PROGRAM prgMotionRow
VAR
		tStationNumberIndex: UINT;	
		tNumElementsPerScreen: UINT;
		tScreenElementsPerPage: UINT;
		tTrueStationIndex: UINT;
		tSizeOfMotionRow: UINT;
		tSizeOfMotionRowButtons: UINT;
		retval: UDINT;
		btnNext:R_TRIG;
		btnPrev:R_TRIG;
		
		btnNextRow:R_TRIG;
		btnPrevRow:R_TRIG;
		tSingleRowOffset: UINT;
		
	tSingleRowOffsettest: UINT;
	tSingleRowOffsettestbtns: UINT;
	tSizeOfButtonsLen: UINT;
	tSizeOfRowSingleLens: UINT;
	
	tSingleRowOffsetFactor:UINT;
	tSingleRowOffsetPointer: UINT;
END_VAR

//call logic for Motion screen using motion Rows

//select station on HMI
actPageControl();

//calculate screen range
actCalcScreenNumber();

//call manual screen rows
actCallMotionScreen();

//calculate screen range
actCalcMotionRowPosn();

//calculate page title
actCalcPageTitle();

ACTION actCalcMotionRowPosn:
//calaculate station index for pages
tTrueStationIndex := tStationNumberIndex + ((tScreenElementsPerPage * gHMIData.gActivePageNumber) -  tScreenElementsPerPage);


tSingleRowOffsetPointer := (tSingleRowOffsetFactor *  gHMIDataConst.gNumberElementsPerRow) - gHMIDataConst.gNumberElementsPerRow;
tSingleRowOffsetPointer := tSingleRowOffsetPointer + gHMIDataConst.gNumberElementsPerRow;

//test for singular row change
tTrueStationIndex := tTrueStationIndex + tSingleRowOffsetPointer;

//calculate offset for row x
gHMIData.gRowElementOffset[1]:= tTrueStationIndex + ((gHMIDataConst.gNumberElementsPerRow * 1) - gHMIDataConst.gNumberElementsPerRow);
gHMIData.gRowElementOffset[2]:= tTrueStationIndex + ((gHMIDataConst.gNumberElementsPerRow * 2) - gHMIDataConst.gNumberElementsPerRow);
gHMIData.gRowElementOffset[3]:= tTrueStationIndex + ((gHMIDataConst.gNumberElementsPerRow * 3) - gHMIDataConst.gNumberElementsPerRow);
gHMIData.gRowElementOffset[4]:= tTrueStationIndex + ((gHMIDataConst.gNumberElementsPerRow * 4) - gHMIDataConst.gNumberElementsPerRow);
gHMIData.gRowElementOffset[5]:= tTrueStationIndex + ((gHMIDataConst.gNumberElementsPerRow * 5) - gHMIDataConst.gNumberElementsPerRow);
gHMIData.gRowElementOffset[6]:= tTrueStationIndex + ((gHMIDataConst.gNumberElementsPerRow * 6) - gHMIDataConst.gNumberElementsPerRow);
gHMIData.gRowElementOffset[7]:= tTrueStationIndex + ((gHMIDataConst.gNumberElementsPerRow * 7) - gHMIDataConst.gNumberElementsPerRow);
gHMIData.gRowElementOffset[8]:= tTrueStationIndex + ((gHMIDataConst.gNumberElementsPerRow * 8) - gHMIDataConst.gNumberElementsPerRow);
gHMIData.gRowElementOffset[9]:= tTrueStationIndex + ((gHMIDataConst.gNumberElementsPerRow * 9) - gHMIDataConst.gNumberElementsPerRow);


//move to global to be picked up by each row
gHMIMotionRows.gMotionRows.gMotionRow1.IndexLocation := gHMIData.gRowElementOffset[1];
gHMIMotionRows.gMotionRows.gMotionRow2.IndexLocation := gHMIData.gRowElementOffset[2];
gHMIMotionRows.gMotionRows.gMotionRow3.IndexLocation := gHMIData.gRowElementOffset[3];
gHMIMotionRows.gMotionRows.gMotionRow4.IndexLocation := gHMIData.gRowElementOffset[4];
gHMIMotionRows.gMotionRows.gMotionRow5.IndexLocation := gHMIData.gRowElementOffset[5];
gHMIMotionRows.gMotionRows.gMotionRow6.IndexLocation := gHMIData.gRowElementOffset[6];
gHMIMotionRows.gMotionRows.gMotionRow7.IndexLocation := gHMIData.gRowElementOffset[7];
gHMIMotionRows.gMotionRows.gMotionRow8.IndexLocation := gHMIData.gRowElementOffset[8];
gHMIMotionRows.gMotionRows.gMotionRow9.IndexLocation := gHMIData.gRowElementOffset[9];
END_ACTION

ACTION actCalcPageTitle:
//get the page number index relating the group of motions displayed
gHMIData.gManualScreenTitle := tStationNumberIndex + gHMIData.gActivePageNumber;

//10001 = station 1, page 1
//10002 = station 1, page 2

//20001 = station 1, page 1
//etc

//assign text in textlist ManualPageTitle
END_ACTION

ACTION actCalcScreenNumber:
//create number for station
tStationNumberIndex := gHMIData.gActiveStationNumber * 10000;

//calculate number of elements per screen
tNumElementsPerScreen := gHMIDataConst.gNumberRowsPerPage * gHMIDataConst.gNumberElementsPerRow;

//calculate screen per page index
tScreenElementsPerPage := tNumElementsPerScreen  * 1;
END_ACTION

ACTION actCallMotionScreen:
//calculate byte offset - motions
tSizeOfMotionRow		:= gHMIData.gActivePageNumber * SIZEOF(gHMIMotionRows.gMotionRows);
tSizeOfMotionRow 		:= tSizeOfMotionRow - SIZEOF(gHMIMotionRows.gMotionRows);

//test for singular row changes
tSizeOfRowSingleLens := SIZEOF(typeMotionRow); //typ 153 bytes
tSizeOfMotionRow := tSizeOfMotionRow + (tSingleRowOffsetFactor * tSizeOfRowSingleLens) ;


//calculate byte offset - buttons
tSizeOfMotionRowButtons := gHMIData.gActivePageNumber * SIZEOF(gHMIMotionRows.gMotionRowButtons);
tSizeOfMotionRowButtons := tSizeOfMotionRowButtons - SIZEOF(gHMIMotionRows.gMotionRowButtons);

//test for singular row changes
tSizeOfButtonsLen := SIZEOF(typeMotionRowButtons); // typ 83 bytes
tSizeOfMotionRowButtons := tSizeOfMotionRowButtons + (tSingleRowOffsetFactor * tSizeOfButtonsLen);

//move data based on station and page number
//Move feedback indicator data
//Move Button BOOL state back adr(S1_Global.MotionRow)
IF gHMIData.gStationSelected[1] THEN
	retval := memcpy(	destAddr:=	ADR(gHMIMotionRows.gMotionRows),
						srcAddr:=	ADR(S1_Global.station.MotionRow) + tSizeOfMotionRow,
						n:=			SIZEOF(gHMIMotionRows.gMotionRows)
						);
						
	retval := memcpy(	destAddr:=	ADR(S1_Global.station.MotionRowBtn) + tSizeOfMotionRowButtons,
						srcAddr:=	ADR(gHMIMotionRows.gMotionRowButtons),
						n:=			SIZEOF(gHMIMotionRows.gMotionRowButtons)
						);
END_IF

IF gHMIData.gStationSelected[2] THEN
	retval := memcpy(	destAddr:=	ADR(gHMIMotionRows.gMotionRows),
						srcAddr:=	ADR(S2_Global.station.MotionRow) + tSizeOfMotionRow,
						n:=			SIZEOF(gHMIMotionRows.gMotionRows)
						);
						
	retval := memcpy(	destAddr:=	ADR(S2_Global.station.MotionRowBtn) + tSizeOfMotionRowButtons,
						srcAddr:=	ADR(gHMIMotionRows.gMotionRowButtons),
						n:=			SIZEOF(gHMIMotionRows.gMotionRowButtons)
						);
END_IF

IF gHMIData.gStationSelected[3] THEN
	retval := memcpy(	destAddr:=	ADR(gHMIMotionRows.gMotionRows),
						srcAddr:=	ADR(S3_Global.station.MotionRow) + tSizeOfMotionRow,
						n:=			SIZEOF(gHMIMotionRows.gMotionRows)
						);
						
	retval := memcpy(	destAddr:=	ADR(S3_Global.station.MotionRowBtn) + tSizeOfMotionRowButtons,
						srcAddr:=	ADR(gHMIMotionRows.gMotionRowButtons),
						n:=			SIZEOF(gHMIMotionRows.gMotionRowButtons)
						);
END_IF

IF gHMIData.gStationSelected[4] THEN
	retval := memcpy(	destAddr:=	ADR(gHMIMotionRows.gMotionRows),
						srcAddr:=	ADR(S4_Global.station.MotionRow) + tSizeOfMotionRow,
						n:=			SIZEOF(gHMIMotionRows.gMotionRows)
						);
						
	retval := memcpy(	destAddr:=	ADR(S4_Global.station.MotionRowBtn) + tSizeOfMotionRowButtons,
						srcAddr:=	ADR(gHMIMotionRows.gMotionRowButtons),
						n:=			SIZEOF(gHMIMotionRows.gMotionRowButtons)
						);
END_IF

IF gHMIData.gStationSelected[5] THEN
	retval := memcpy(	destAddr:=	ADR(gHMIMotionRows.gMotionRows),
						srcAddr:=	ADR(S5_Global.station.MotionRow) + tSizeOfMotionRow,
						n:=			SIZEOF(gHMIMotionRows.gMotionRows)
						);
						
	retval := memcpy(	destAddr:=	ADR(S5_Global.station.MotionRowBtn) + tSizeOfMotionRowButtons,
						srcAddr:=	ADR(gHMIMotionRows.gMotionRowButtons),
						n:=			SIZEOF(gHMIMotionRows.gMotionRowButtons)
						);
END_IF

IF gHMIData.gStationSelected[6] THEN
	retval := memcpy(	destAddr:=	ADR(gHMIMotionRows.gMotionRows),
						srcAddr:=	ADR(S6_Global.station.MotionRow) + tSizeOfMotionRow,
						n:=			SIZEOF(gHMIMotionRows.gMotionRows)
						);
						
	retval := memcpy(	destAddr:=	ADR(S6_Global.station.MotionRowBtn) + tSizeOfMotionRowButtons,
						srcAddr:=	ADR(gHMIMotionRows.gMotionRowButtons),
						n:=			SIZEOF(gHMIMotionRows.gMotionRowButtons)
						);
END_IF
END_ACTION

ACTION actPageControl:
//imply TRIG call
btnNext(clk:=gHMIButtons.btnNextPage);
btnPrev(clk:=gHMIButtons.btnPrevPage);

//imply TRIG call
btnNextRow(clk:=gHMIButtons.btnPlus1Row); 
btnPrevRow(clk:=gHMIButtons.btnNeg1Row);

//next page
IF btnNext.Q THEN
	gHMIData.gActivePageNumber := gHMIData.gActivePageNumber + 1;
	
	//reset single offset
	tSingleRowOffsetFactor := 0;
END_IF

//previous page
IF btnPrev.Q THEN
	gHMIData.gActivePageNumber := gHMIData.gActivePageNumber - 1;
	
	//reset single offset
	tSingleRowOffsetFactor := 0;
END_IF

//apply limits
IF gHMIData.gActivePageNumber < 1 THEN
	gHMIData.gActivePageNumber := 1;
END_IF

//apply limits
IF gHMIData.gActivePageNumber > gHMIData.gMaxPageNumber THEN
	gHMIData.gActivePageNumber := gHMIData.gMaxPageNumber;
END_IF

//station 1 control
IF gHMIData.gStationSelected[1] THEN
	gHMIData.gMaxPageNumber := S1_Global.station.Data.NumberOfPages;
END_IF

//station 2 control
IF gHMIData.gStationSelected[2] THEN
	gHMIData.gMaxPageNumber := S2_Global.station.Data.NumberOfPages;
END_IF

//station 3 control
IF gHMIData.gStationSelected[3] THEN
	gHMIData.gMaxPageNumber := S3_Global.station.Data.NumberOfPages;
END_IF

//station 4 control
IF gHMIData.gStationSelected[4] THEN
	gHMIData.gMaxPageNumber := S4_Global.station.Data.NumberOfPages;
END_IF

//station 5 control
IF gHMIData.gStationSelected[5] THEN
	gHMIData.gMaxPageNumber := S5_Global.station.Data.NumberOfPages;
END_IF

//station 6 control
IF gHMIData.gStationSelected[6] THEN
	gHMIData.gMaxPageNumber := S6_Global.station.Data.NumberOfPages;
END_IF

//calc single row offset
//tSingleRowOffset
IF btnNextRow.Q THEN
tSingleRowOffsetFactor := tSingleRowOffsetFactor +1;
END_IF

IF btnPrevRow.Q THEN
tSingleRowOffsetFactor := tSingleRowOffsetFactor - 1;
END_IF

//single row cleanup
IF tSingleRowOffsetFactor >= 65535 THEN
	tSingleRowOffsetFactor := 0;
END_IF
END_ACTION

END_PROGRAM

(* stored: Version 1.1.0.1, ProductVersion 3.1.4024.11
   POU prgMotionRow: Id {4ecda869-418e-4b2d-994d-c4c6ccf53283}, SpecialFunc None
   Action actCalcMotionRowPosn: Id {d052a485-2ab5-4274-9ad1-f666fbdc1383}
   Action actCalcPageTitle: Id {904b6009-924e-4962-82c3-1f501316d522}
   Action actCalcScreenNumber: Id {6c34dbe5-12b3-4058-a71b-5a6feb4de7c0}
   Action actCallMotionScreen: Id {7fde1ebb-b0f7-4572-8651-feb24111554c}
   Action actPageControl: Id {30c64ed5-f661-4d65-b1ea-51ade9043dc1} *)
